Yaskawa INFORM job: R1_W23(-90,90)(KAMERA)KM-OK.JBI

/JOB
//NAME R1_W23(-90,90)(KAMERA)KM-OK
///FOLDERNAME SCIANA-NOWY-R2-KM
//POS
///NPOS 52,52,0,5,0,0
///TOOL 0
///POSTYPE PULSE
///PULSE
C00000=88675,32979,-24114,16557,98507,-59299
C00001=17025,-102762,-106901,19715,68975,-69577
C00002=8925,32874,-5917,15999,81635,-77978
C00003=6731,-8881,-33435,24026,63611,-65551
C00004=162577,-11667,-36907,20520,58968,-63561
C00005=203471,-60021,-49027,-10079,38921,-46363
C00006=203097,-42314,-31129,-10161,36999,-46322
C00007=203097,-42314,-31129,-10161,36999,-46322
C00008=203578,-40766,-30177,-10560,37265,-46086
C00009=203097,-42314,-31129,-10161,36999,-46322
C00010=203097,-42140,-30574,-10220,36752,-46288
C00011=203097,-42314,-31129,-10161,36999,-46322
C00012=191626,-47104,-40278,-407,41031,-52175
C00013=139702,-43395,-38511,37598,53562,-75420
C00014=142881,-40428,-32128,37248,50251,-75168
C00015=144416,-39055,-29758,36884,48980,-74892
C00016=144416,-38687,-28536,37177,48526,-75095
C00017=144416,-39055,-29758,36884,48980,-74892
C00018=145553,-38396,-29341,36271,48560,-74454
C00019=144416,-39055,-29758,36884,48980,-74892
C00020=137911,-53706,-46488,38566,54043,-76145
C00021=153698,-43990,-63296,-25548,87073,-75741
C00022=156931,-42686,-47572,-39341,82743,-73197
C00023=147752,-38541,-33018,-46313,75351,-74633
C00024=147235,-38379,-32306,-46377,75472,-74522
C00025=147235,-38038,-31017,-46485,75038,-74313
C00026=147235,-38379,-32306,-46377,75472,-74522
C00027=146168,-39057,-32734,-46256,74860,-74755
C00028=147235,-38379,-32306,-46377,75472,-74522
C00029=152316,-36319,-36213,-46469,79906,-74572
C00030=151626,-33267,-34218,-46339,79789,-74852
C00031=146248,-37226,-30843,-46229,74106,-74780
C00032=146248,-37226,-30843,-46229,74106,-74780
C00033=145623,-37613,-31090,-46152,73751,-74917
C00034=146248,-37226,-30843,-46229,74106,-74780
C00035=146248,-37050,-30186,-46289,73885,-74672
C00036=146248,-37226,-30843,-46229,74106,-74780
C00037=155476,-32068,-36597,-46659,83246,-74625
C00038=172432,-59305,-63154,-24054,64023,-64136
C00039=203471,-60021,-49027,-10079,38921,-46363
C00040=211074,-47059,-33081,-17754,36709,-41881
C00041=188633,-22668,-17345,4103,37677,-54473
C00042=176443,2386,1899,14891,40129,-60743
C00043=172652,-6496,-11395,16872,44320,-61929
C00044=219374,-84444,-80719,-20673,48228,-40195
C00045=138726,-34606,-61985,-42967,96530,-79520
C00046=142080,-58876,-49418,-42986,83059,-72427
C00047=128671,-45230,-35751,-42125,64007,-78461
C00048=126309,8548,3685,-40494,65278,-80277
C00049=125516,41789,35777,-41114,62867,-79626
C00050=129180,33981,13394,-39638,72105,-81689
C00051=131035,15732,-13271,-39136,78432,-83284
BC00000=287186,1180734,1073595
BC00001=5669,1187291,1073594
BC00002=21598,1304301,1073588
BC00003=153725,1258504,1073599
BC00004=397442,1187982,1073599
BC00005=397442,1061622,1073599
BC00006=397442,1061621,1073596
BC00007=397442,1061621,1073596
BC00008=397442,1061621,1073596
BC00009=397442,1061621,1073596
BC00010=397442,1061621,1073596
BC00011=397442,1061621,1073596
BC00012=389747,1061621,1073596
BC00013=313972,1061621,1073596
BC00014=313972,1061621,1073596
BC00015=313972,1061621,1073596
BC00016=313972,1061621,1073596
BC00017=313972,1061621,1073596
BC00018=313972,1061621,1073596
BC00019=313972,1061621,1073596
BC00020=313972,1061621,1073596
BC00021=241083,1061621,1073656
BC00022=226163,1061621,1073596
BC00023=226163,1061621,1073596
BC00024=226163,1061621,1073596
BC00025=226163,1061621,1073596
BC00026=226163,1061621,1073596
BC00027=226163,1061621,1073596
BC00028=226163,1061621,1073596
BC00029=226163,1061621,1073596
BC00030=226163,1136276,1073596
BC00031=226163,1136276,1073596
BC00032=226163,1136276,1073596
BC00033=226163,1136276,1073596
BC00034=226163,1136276,1073596
BC00035=226163,1136276,1073596
BC00036=226163,1136276,1073596
BC00037=226163,1136276,1073596
BC00038=312007,1098860,1073598
BC00039=397442,1061622,1073599
BC00040=397442,1053865,1073599
BC00041=397445,1053866,1073597
BC00042=397442,1053865,1073599
BC00043=397442,1053865,1073599
BC00044=397442,1053865,1073599
BC00045=194089,1142515,1073599
BC00046=194089,1142515,1073599
BC00047=194089,1142515,1073599
BC00048=194089,1142515,1073599
BC00049=194089,1142515,1073599
BC00050=194089,1142515,1073599
BC00051=194089,1142515,1073599
///POSTYPE BASE
///RECTAN
///RCONF 0,0,0,0,0,0,0,0,0,0,0,0,0,0,0,0,0,0,0,0,0,0,0,0
P00006=0.222,-3.123,-1.508,0.0000,0.0000,0.0000
P00021=-0.225,-6.128,-0.405,0.0000,0.0000,0.0000
P00022=0.222,-3.123,-1.508,0.0000,0.0000,0.0000
P00023=0.143,-0.036,0.682,0.0000,0.0000,0.0000
P00024=0.145,-0.552,1.326,0.0000,0.0000,0.0000
//INST
///DATE 2024/07/29 11:35
///ATTR SC,RW
///GROUP1 RB1,BS1
NOP
'r1_W23(-90,90)(kamera)
'Path W869
SFTOF
MOVJ C00000 BC00000 VJ=100.00
MOVJ C00001 BC00001 VJ=100.00
MOVJ C00002 BC00002 VJ=100.00
CALL JOB:CLEAN-R1_KM_NEW_SCIANA
MOVJ C00003 BC00003 VJ=100.00
MOVJ C00004 BC00004 VJ=100.00
MOVJ C00005 BC00005 VJ=100.00
MOVJ C00006 BC00006 VJ=100.00
'POMIAR
MOVL C00007 BC00007 V=60.0
REFP 3 C00008 BC00008
CALL JOB:SEARCH-R1
SET P021 P006
SFTON P021
MOVL C00009 BC00009 V=60.0
REFP 3 C00010 BC00010
CALL JOB:SEARCH-R1
SET P021 P006
SFTON P021
MOVL C00011 BC00011 V=60.0
MOVJ C00012 BC00012 VJ=100.00
SFTOF
MOVJ C00013 BC00013 VJ=100.00
MOVJ C00014 BC00014 VJ=100.00
MOVL C00015 BC00015 V=60.0
REFP 3 C00016 BC00016
CALL JOB:SEARCH-R1
SET P022 P006
SFTON P022
MOVL C00017 BC00017 V=60.0
REFP 3 C00018 BC00018
CALL JOB:SEARCH-R1
SET P022 P006
SFTON P022
MOVL C00019 BC00019 V=60.0
MOVJ C00020 BC00020 VJ=100.00
SFTOF
MOVJ C00021 BC00021 VJ=100.00
MOVJ C00022 BC00022 VJ=100.00
MOVJ C00023 BC00023 VJ=100.00
MOVL C00024 BC00024 V=60.0
REFP 3 C00025 BC00025
CALL JOB:SEARCH-R1
SET P023 P006
SFTON P023
MOVL C00026 BC00026 V=60.0
REFP 3 C00027 BC00027
CALL JOB:SEARCH-R1
SET P023 P006
SFTON P023
MOVL C00028 BC00028 V=60.0
MOVJ C00029 BC00029 VJ=100.00
SFTOF
MOVJ C00030 BC00030 VJ=100.00
MOVJ C00031 BC00031 VJ=100.00
MOVL C00032 BC00032 V=60.0
REFP 3 C00033 BC00033
CALL JOB:SEARCH-R1
SET P024 P006
SFTON P024
MOVL C00034 BC00034 V=60.0
REFP 3 C00035 BC00035
CALL JOB:SEARCH-R1
SET P024 P006
SFTON P024
MOVL C00036 BC00036 V=60.0
MOVJ C00037 BC00037 VJ=100.00
MOVJ C00038 BC00038 VJ=100.00
SFTOF
MOVJ C00039 BC00039 VJ=100.00
SFTON P021
MOVJ C00040 BC00040 VJ=100.00
MACRO1 MJ#(0) ARGF9
ARCON
SFTON P022
MOVL C00041 BC00041 V=9.2
MOVL C00042 BC00042 V=9.2
ARCOF
SFTOF
MOVL C00043 BC00043 V=166.7
MOVJ C00044 BC00044 VJ=100.00
MOVJ C00045 BC00045 VJ=100.00
'SPOINA2
MOVJ C00046 BC00046 VJ=100.00
SFTON P024
MOVJ C00047 BC00047 VJ=15.00
MACRO1 MJ#(0) ARGF9
ARCON
SFTON P023
MOVL C00048 BC00048 V=9.2
MOVL C00049 BC00049 V=9.2
ARCOF
SFTOF
MOVJ C00050 BC00050 VJ=100.00
MOVJ C00051 BC00051 VJ=100.00
END
